PROGRAM pump_manager
VAR
	//Repeat for each pump?
	u_3112_enable: BOOL;
	u_3112_idle_request: BOOL;
	u_3112_cip_request: BOOL;
	u_3112_manual_request: BOOL;
	u_3112_stop_request: BOOL;
	u_3112_intlk: BOOL;
	u_3112_maint_request: BOOL;
	u_3112_idle_speed_request: REAL;
	u_3112_setpoint_request: REAL;
	u_3112_cip_speed_request: REAL;
	u_3112_manual_speed_request: REAL;
	u_3112_maint_speed_request: REAL;
	
	u_3212_enable: BOOL;
	u_3212_idle_request: BOOL;
	u_3212_cip_request: BOOL;
	u_3212_manual_request: BOOL;
	u_3212_stop_request: BOOL;
	u_3212_intlk: BOOL;
	u_3212_maint_request: BOOL;
	u_3212_idle_speed_request: REAL;
	u_3212_setpoint_request: REAL;
	u_3212_cip_speed_request: REAL;
	u_3212_manual_speed_request: REAL;
	u_3212_maint_speed_request: REAL;
	
	u_3312_enable: BOOL;
	u_3312_idle_request: BOOL;
	u_3312_cip_request: BOOL;
	u_3312_manual_request: BOOL;
	u_3312_stop_request: BOOL;
	u_3312_intlk: BOOL;
	u_3312_maint_request: BOOL;
	u_3312_idle_speed_request: REAL;
	u_3312_speed_request: REAL;
	u_3312_cip_speed_request: REAL;
	u_3312_manual_speed_request: REAL;
	u_3312_maint_speed_request: REAL;
	
	u_3405_enable: BOOL;
	u_3405_idle_request: BOOL;
	u_3405_cip_request: BOOL;
	u_3405_manual_request: BOOL;
	u_3405_stop_request: BOOL;
	u_3405_intlk: BOOL;
	u_3405_maint_request: BOOL;
	u_3405_idle_speed_request: REAL;
	u_3405_speed_request: REAL;
	u_3405_cip_speed_request: REAL;
	u_3405_manual_speed_request: REAL;
	u_3405_maint_speed_request: REAL;
	
	u_3160_enable: BOOL;
	u_3160_idle_request: BOOL;
	u_3160_cip_request: BOOL;
	u_3160_manual_request: BOOL;
	u_3160_stop_request: BOOL;
	u_3160_intlk: BOOL;
	u_3160_maint_request: BOOL;
	u_3160_idle_speed_request: REAL;
	u_3160_speed_request: REAL;
	u_3160_cip_speed_request: REAL;
	u_3160_manual_speed_request: REAL;
	u_3160_maint_speed_request: REAL;
	
	u_3260_enable: BOOL;
	u_3260_idle_request: BOOL;
	u_3260_cip_request: BOOL;
	u_3260_manual_request: BOOL;
	u_3260_stop_request: BOOL;
	u_3260_intlk: BOOL;
	u_3260_maint_request: BOOL;
	u_3260_idle_speed_request: REAL;
	u_3260_speed_request: REAL;
	u_3260_cip_speed_request: REAL;
	u_3260_manual_speed_request: REAL;
	u_3260_maint_speed_request: REAL;
	
	u_3360_enable: BOOL;
	u_3360_idle_request: BOOL;
	u_3360_cip_request: BOOL;
	u_3360_manual_request: BOOL;
	u_3360_stop_request: BOOL;
	u_3360_intlk: BOOL;
	u_3360_maint_request: BOOL;
	u_3360_idle_speed_request: REAL;
	u_3360_speed_request: REAL;
	u_3360_cip_speed_request: REAL;
	u_3360_manual_speed_request: REAL;
	u_3360_maint_speed_request: REAL;
	
	
	gen_alm_active: BOOL;
	ed_routine_idle: BOOL;
	ed_routine_cip: BOOL;
	//ed_routine_manual: BOOL;
	ed_routine_maint: BOOL;
	
	u_3370_enable: BOOL;
	u_3370_idle_request: BOOL;
	u_3370_cip_request: BOOL;
	u_3370_manual_request: BOOL;
	u_3370_stop_request: BOOL;
	u_3370_intlk: BOOL;
	u_3370_maint_request: BOOL;
	u_3370_idle_speed_request: REAL;
	u_3370_speed_request: REAL;
	u_3370_cip_speed_request: REAL;
	u_3370_manual_speed_request: REAL;
	u_3370_maint_speed_request: REAL;
	u_3312_setpoint_request: REAL;
	u_3405_setpoint_request: REAL;
	u_3112_pid_reset: BOOL;
	u_3112_ons: R_TRIG;
	u_3312_pid_reset: BOOL;
	u_3312_ons: R_TRIG;
	u_3212_ons: R_TRIG;
	u_3212_pid_reset: BOOL;
	u_3405_ons: R_TRIG;
	u_3405_pid_reset: BOOL;
	u_3370_setpoint_request: LREAL;
	u_3370_ons: R_TRIG;
	u_3370_pid_reset: BOOL;
END_VAR
VAR // added by the converter: edge detectors and wires of the graphical bodies
    _w1, _w2, _w3, _w4, _w5, _w6, _w7, _w8, _w9, _w10 : BOOL;
END_VAR

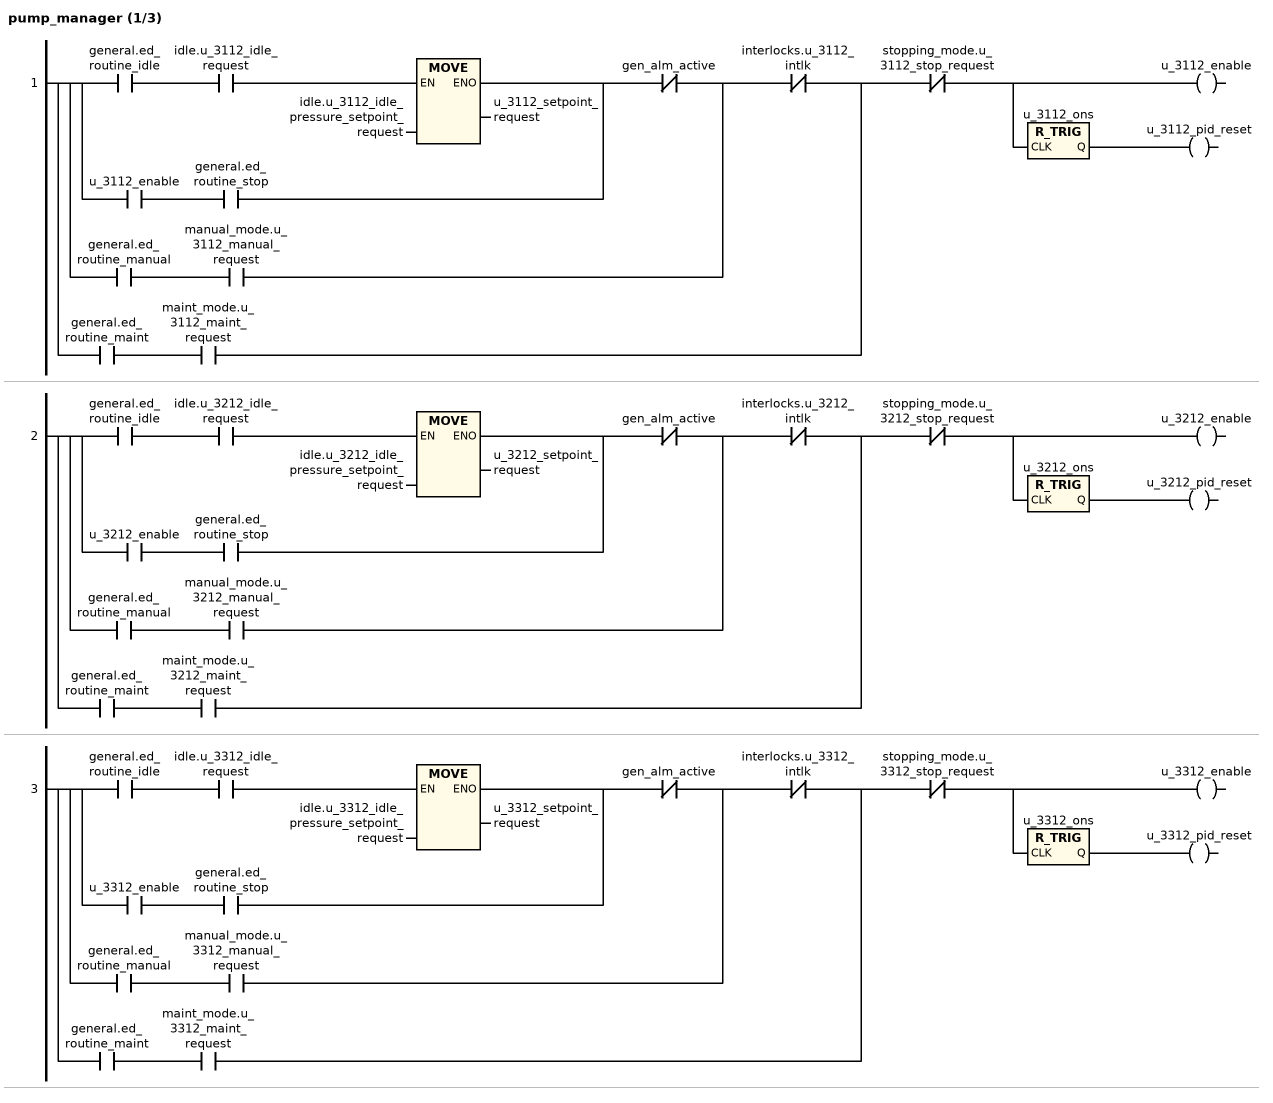
// NETWORK 1
_w1 := general.ed_routine_idle AND idle.u_3112_idle_request;
IF _w1 THEN u_3112_setpoint_request := idle.u_3112_idle_pressure_setpoint_request; END_IF
_w2 := (((_w1 OR u_3112_enable AND general.ed_routine_stop) AND NOT gen_alm_active OR general.ed_routine_manual AND manual_mode.u_3112_manual_request) AND NOT interlocks.u_3112_intlk OR general.ed_routine_maint AND maint_mode.u_3112_maint_request) AND NOT stopping_mode.u_3112_stop_request;
u_3112_enable := _w2;
u_3112_ons(CLK := _w2); // R_TRIG
u_3112_pid_reset := u_3112_ons.Q;

// NETWORK 2
_w3 := general.ed_routine_idle AND idle.u_3212_idle_request;
IF _w3 THEN u_3212_setpoint_request := idle.u_3212_idle_pressure_setpoint_request; END_IF
_w4 := (((_w3 OR u_3212_enable AND general.ed_routine_stop) AND NOT gen_alm_active OR general.ed_routine_manual AND manual_mode.u_3212_manual_request) AND NOT interlocks.u_3212_intlk OR general.ed_routine_maint AND maint_mode.u_3212_maint_request) AND NOT stopping_mode.u_3212_stop_request;
u_3212_enable := _w4;
u_3212_ons(CLK := _w4); // R_TRIG
u_3212_pid_reset := u_3212_ons.Q;

// NETWORK 3
_w5 := general.ed_routine_idle AND idle.u_3312_idle_request;
IF _w5 THEN u_3312_setpoint_request := idle.u_3312_idle_pressure_setpoint_request; END_IF
_w6 := (((_w5 OR u_3312_enable AND general.ed_routine_stop) AND NOT gen_alm_active OR general.ed_routine_manual AND manual_mode.u_3312_manual_request) AND NOT interlocks.u_3312_intlk OR general.ed_routine_maint AND maint_mode.u_3312_maint_request) AND NOT stopping_mode.u_3312_stop_request;
u_3312_enable := _w6;
u_3312_ons(CLK := _w6); // R_TRIG
u_3312_pid_reset := u_3312_ons.Q;

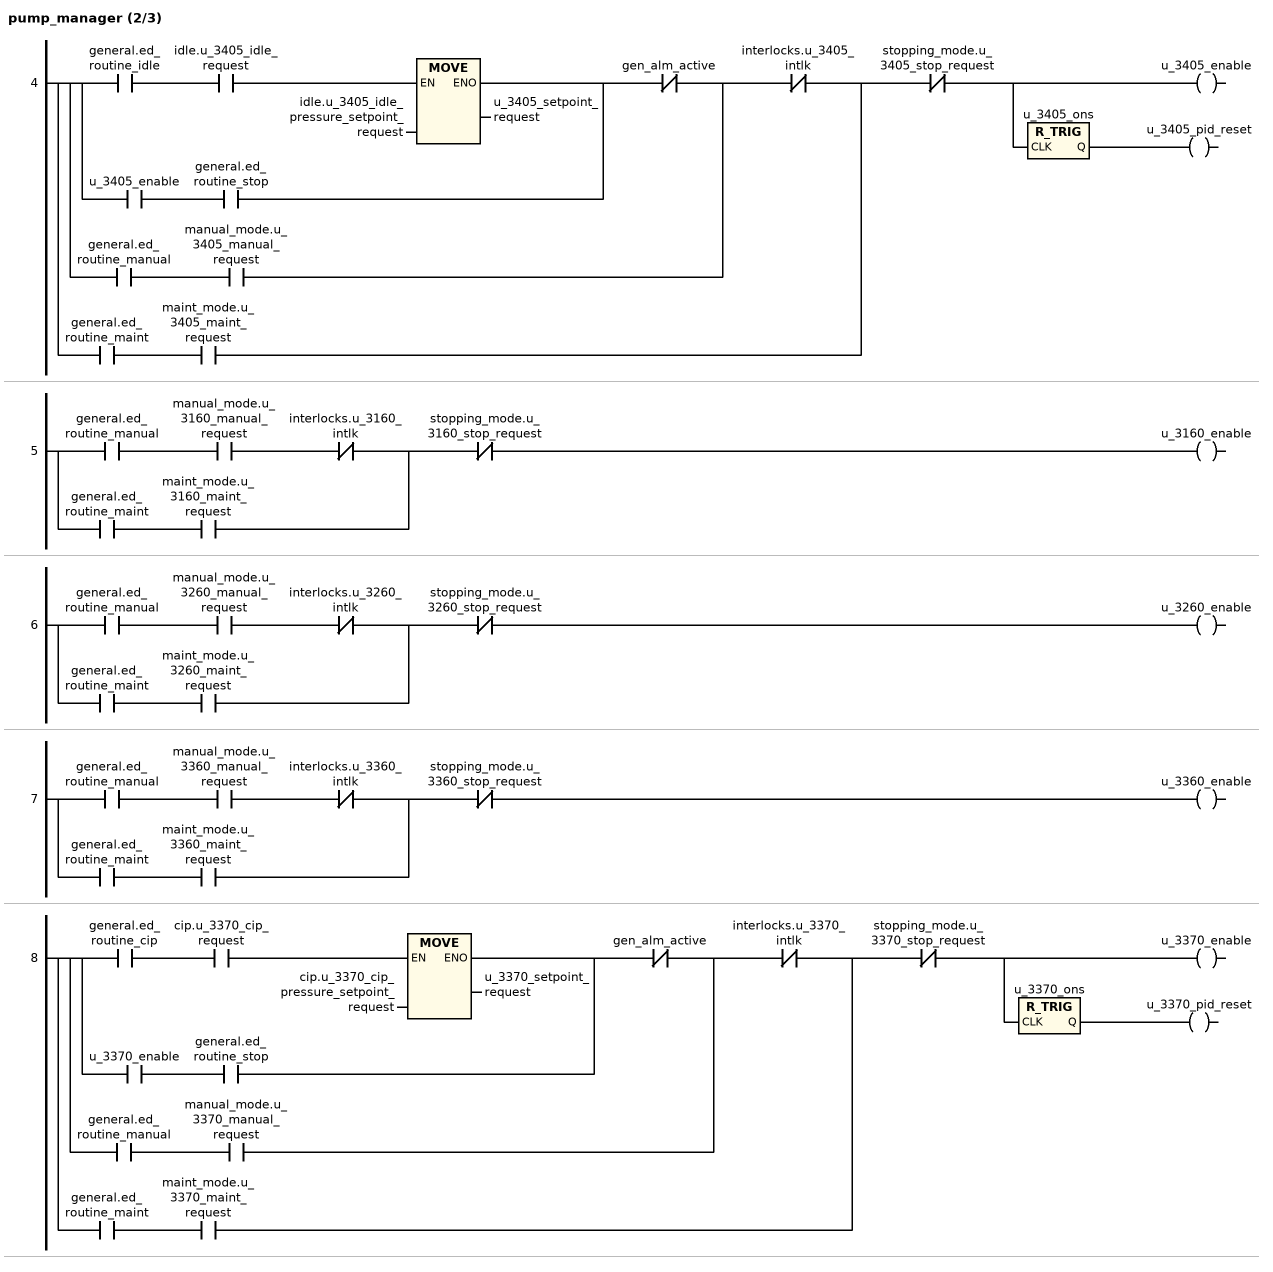
// NETWORK 4
_w7 := general.ed_routine_idle AND idle.u_3405_idle_request;
IF _w7 THEN u_3405_setpoint_request := idle.u_3405_idle_pressure_setpoint_request; END_IF
_w8 := (((_w7 OR u_3405_enable AND general.ed_routine_stop) AND NOT gen_alm_active OR general.ed_routine_manual AND manual_mode.u_3405_manual_request) AND NOT interlocks.u_3405_intlk OR general.ed_routine_maint AND maint_mode.u_3405_maint_request) AND NOT stopping_mode.u_3405_stop_request;
u_3405_enable := _w8;
u_3405_ons(CLK := _w8); // R_TRIG
u_3405_pid_reset := u_3405_ons.Q;

// NETWORK 5
u_3160_enable := (general.ed_routine_manual AND manual_mode.u_3160_manual_request AND NOT interlocks.u_3160_intlk OR general.ed_routine_maint AND maint_mode.u_3160_maint_request) AND NOT stopping_mode.u_3160_stop_request;

// NETWORK 6
u_3260_enable := (general.ed_routine_manual AND manual_mode.u_3260_manual_request AND NOT interlocks.u_3260_intlk OR general.ed_routine_maint AND maint_mode.u_3260_maint_request) AND NOT stopping_mode.u_3260_stop_request;

// NETWORK 7
u_3360_enable := (general.ed_routine_manual AND manual_mode.u_3360_manual_request AND NOT interlocks.u_3360_intlk OR general.ed_routine_maint AND maint_mode.u_3360_maint_request) AND NOT stopping_mode.u_3360_stop_request;

// NETWORK 8
_w9 := general.ed_routine_cip AND cip.u_3370_cip_request;
IF _w9 THEN u_3370_setpoint_request := cip.u_3370_cip_pressure_setpoint_request; END_IF
_w10 := (((_w9 OR u_3370_enable AND general.ed_routine_stop) AND NOT gen_alm_active OR general.ed_routine_manual AND manual_mode.u_3370_manual_request) AND NOT interlocks.u_3370_intlk OR general.ed_routine_maint AND maint_mode.u_3370_maint_request) AND NOT stopping_mode.u_3370_stop_request;
u_3370_enable := _w10;
u_3370_ons(CLK := _w10); // R_TRIG
u_3370_pid_reset := u_3370_ons.Q;

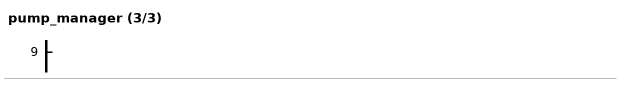
// NETWORK 9

END_PROGRAM

(* stored: Version 1.1.0.1, ProductVersion 3.1.4024.12
   POU pump_manager: Id {3b5ad67c-a464-4c74-9317-fc4708b2e954}, SpecialFunc None *)
